% RSLogix 500 project OVEN LOGIC FINAL.RSS, saved by version 8.30.00.16 %
PROJECT "ABC"    % processor: Bul.1763 MicroLogix 1100 Series B %

PROGRAM FILES
  LAD 2   8 rungs

DATA FILES
  O0 OUTPUT  4 elements
  I1 INPUT  6 elements
  S2 STATUS  66 elements
  B3 BINARY  1 elements
  T4 TIMER  3 elements
  C5 COUNTER  1 elements
  R6 CONTROL  1 elements
  N7 INTEGER  1 elements
  F8 FLOAT  1 elements

LADDER 2
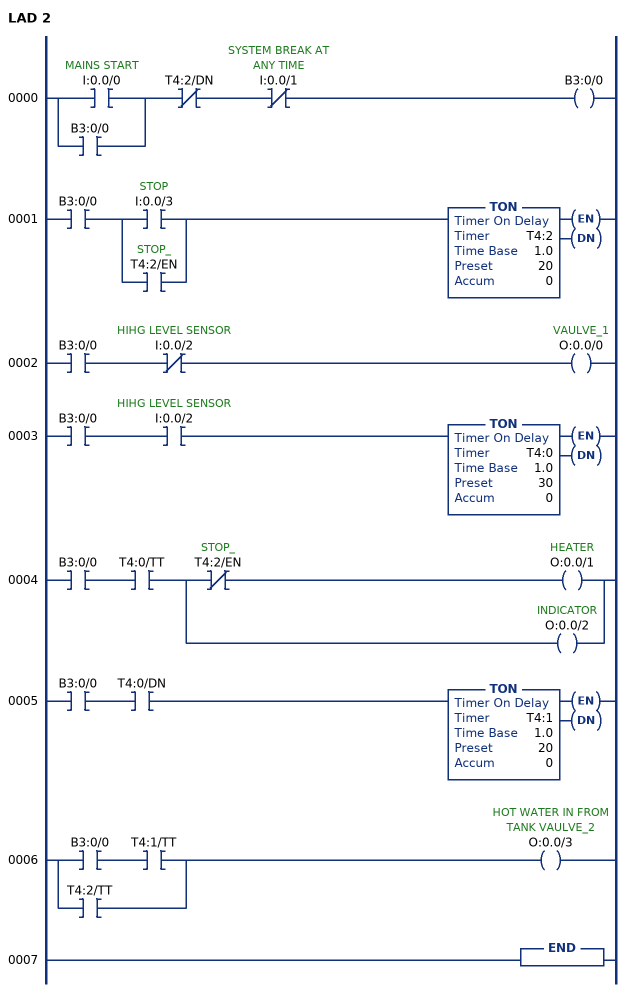
% Rung: 0 %
SOR BST XIC I:0.0/0 NXB XIC B3:0/0 BND XIO T4:2/DN XIO I:0.0/1 OTE B3:0/0 EOR
%   I:0.0/0  START  "MAINS" %
%   I:0.0/1  "SYSTEM BREAK AT ANY TIME" %
% Rung: 1 %
SOR XIC B3:0/0 BST XIC I:0.0/3 NXB XIC T4:2/EN BND TON T4:2 1.0 20 0 EOR
%   I:0.0/3  STOP %
%   T4:2/EN  STOP_ %
% Rung: 2 %
SOR XIC B3:0/0 XIO I:0.0/2 OTE O:0.0/0 EOR
%   I:0.0/2  SENSOR  "HIHG LEVEL" %
%   O:0.0/0  VAULVE_1 %
% Rung: 3 %
SOR XIC B3:0/0 XIC I:0.0/2 TON T4:0 1.0 30 0 EOR
%   I:0.0/2  SENSOR  "HIHG LEVEL" %
% Rung: 4 %
SOR XIC B3:0/0 XIC T4:0/TT BST XIO T4:2/EN OTE O:0.0/1 NXB OTE O:0.0/2 BND EOR
%   T4:2/EN  STOP_ %
%   O:0.0/1  HEATER %
%   O:0.0/2  INDICATOR %
% Rung: 5 %
SOR XIC B3:0/0 XIC T4:0/DN TON T4:1 1.0 20 0 EOR
% Rung: 6 %
SOR BST XIC B3:0/0 XIC T4:1/TT NXB XIC T4:2/TT BND OTE O:0.0/3 EOR
%   O:0.0/3  VAULVE_2  "HOT WATER IN FROM TANK" %
% Rung: 7 %
SOR END EOR

DATA TABLE (non-zero values as saved)
DATA T4
% .PRE .ACC %
% T4:0 % 30 0
% T4:1 % 20 0
% T4:2 % 20 0
